Yaskawa INFORM job: PROFILE_LONG_1.JBI

/JOB
//NAME PROFILE_LONG_1
//POS
///NPOS 12,0,12,1,0,1
///TOOL 0
///POSTYPE PULSE
///PULSE
C00000=-5589,52178,-97239,-514770,62733,92327
C00001=-4560,140303,-79175,-531005,91927,89683
C00002=-5558,118708,-75468,-508549,49962,93238
C00003=-7645,118717,-75287,-507480,49922,93168
C00004=-6978,145152,-75276,-529906,91799,89601
C00005=-7953,54016,-95107,-513369,62240,92134
C00006=-7953,54016,-95107,-513369,62240,92134
C00007=-6997,143668,-75910,-529680,91437,89643
C00008=-7401,116080,-70730,-504099,43492,93399
C00009=-7401,116080,-70730,-504099,43492,93399
C00010=-1581,144226,-75354,-532284,91942,89621
C00011=-2616,57722,-94741,-516813,63920,92341
EC00000=0
EC00001=0
EC00002=0
EC00003=-94441
EC00004=-94441
EC00005=-94441
EC00006=-187105
EC00007=-187105
EC00008=-187105
EC00009=-276069
EC00010=-276069
EC00011=-276069
///POSTYPE BASE
///RECTAN
///RCONF 1,0,0,0,0,0,0,0,0,0,0,0,0,0,0,0,0,0,0,0,0,0,0,0
P00009=1350.000,-150.000,200.000,-180.0000,-45.0000,0.0000
///POSTYPE PULSE
///PULSE
EX00000=0
//INST
///DATE 2023/06/22 13:01
///ATTR SC,RW
///GROUP1 RB1,ST1
NOP
MOVJ P009 EX000 VJ=12.00
MOVJ C00000 EC00000 VJ=12.00
CALL JOB:SPYON
MOVL C00001 EC00001 V=200.0
MOVL C00002 EC00002 V=200.0
CALL JOB:SPYOF
MOVJ C00003 EC00003 VJ=10.00
CALL JOB:SPYON
MOVL C00004 EC00004 V=200.0
MOVL C00005 EC00005 V=200.0
CALL JOB:SPYOF
MOVJ C00006 EC00006 VJ=12.00
CALL JOB:SPYON
MOVL C00007 EC00007 V=200.0
MOVL C00008 EC00008 V=200.0
CALL JOB:SPYOF
MOVJ C00009 EC00009 VJ=10.00
CALL JOB:SPYON
MOVL C00010 EC00010 V=200.0
MOVL C00011 EC00011 V=200.0
CALL JOB:SPYOF
MOVJ P009 EX000 VJ=10.00
END
